# B&R Automation Studio project work
Automation Studio 4.5.2.102

## Configuration Config1

### Task classes (Cpu.sw)
```
Cyclic#1:
  Program <- Program.prg
Binaries: udbdef, TCData, iomap, ashwac, Role, sysconf, arconfig, asfw, User, ashwd
Libraries: Library1
```

## Logical view

Binary libraries used (declarations not repeated): operator, runtime, astime, AsIecCon

### Library Logical/Libraries/Library1 (ANSIC)

#### Library1.fun - Exported functions and function blocks
```iecst
{REDUND_ERROR} FUNCTION_BLOCK FB_Motor (*Функциональный блок для моделирования двигателя*) (*$GROUP=User,$CAT=User,$GROUPICON=User.png,$CATICON=User.png*)
	VAR_INPUT
		u : {REDUND_UNREPLICABLE} REAL;
	END_VAR
	VAR
		dt : REAL;
	END_VAR
	VAR_OUTPUT
		w : {REDUND_UNREPLICABLE} REAL;
		phi : {REDUND_UNREPLICABLE} REAL;
	END_VAR
	VAR
		integrator : {REDUND_UNREPLICABLE} FB_Integrator;
		Tm : {REDUND_UNREPLICABLE} REAL;
		ke : {REDUND_UNREPLICABLE} REAL;
	END_VAR
END_FUNCTION_BLOCK

{REDUND_ERROR} FUNCTION_BLOCK FB_Integrator (*Функциональный блок интегратора*) (*$GROUP=User,$CAT=User,$GROUPICON=User.png,$CATICON=User.png*)
	VAR_INPUT
		in : {REDUND_UNREPLICABLE} REAL;
	END_VAR
	VAR
		dt : REAL;
	END_VAR
	VAR_OUTPUT
		out : {REDUND_UNREPLICABLE} REAL;
	END_VAR
	VAR
		prev_value : REAL;
	END_VAR
END_FUNCTION_BLOCK

{REDUND_ERROR} FUNCTION_BLOCK FB_Controller (*TODO: Add your comment here*) (*$GROUP=User,$CAT=User,$GROUPICON=User.png,$CATICON=User.png*)
	VAR
		dt : REAL; (*шаг расчёта 0.01*)
	END_VAR
	VAR_INPUT
		e_in : {REDUND_UNREPLICABLE} REAL;
	END_VAR
	VAR_OUTPUT
		u_out : {REDUND_UNREPLICABLE} REAL;
	END_VAR
	VAR
		sum : REAL;
		a : REAL;
		k_p : REAL;
		k_i : REAL;
		max_abs_value : REAL;
		iyOld : REAL;
		integrator : FB_Integrator;
	END_VAR
END_FUNCTION_BLOCK
```

#### FB_Motor.c
```c
#include <bur/plctypes.h>
#ifdef __cplusplus
	extern "C"
	{
#endif
	#include "Library1.h"
#ifdef __cplusplus
	};
#endif
/* Функциональный блок для моделирования двигателя */
void FB_Motor(struct FB_Motor* inst)
{

	REAL a = inst->u/inst->ke - inst->w;
	REAL b = a / inst->Tm;

	inst->integrator.in = b;
	FB_Integrator(&inst->integrator);

	inst->w = inst->integrator.out;

}
```

#### FB_Integrator.c
```c
#include <bur/plctypes.h>
#ifdef __cplusplus
	extern "C"
	{
#endif
	#include "Library1.h"
#ifdef __cplusplus
	};
#endif
/* Функциональный блок интегратора */
void FB_Integrator(struct FB_Integrator* inst)
{
	inst->dt = d_t;
	inst->out = inst->dt * inst->in + inst->prev_value;
	inst->prev_value = inst->out;
}
```

#### FB_Controller.c
```c
#include <bur/plctypes.h>
#ifdef __cplusplus
	extern "C"
	{
#endif
	#include "Library1.h"
#ifdef __cplusplus
	};
#endif
/* TODO: Add your comment here */
void FB_Controller(struct FB_Controller* inst)
{
	REAL a = inst->e_in * inst->k_p;
	REAL b = inst->e_in * inst->k_i;

	a = a > inst->max_abs_value ? inst->max_abs_value : a;
	a = a < -inst->max_abs_value ? -inst->max_abs_value : a;

	inst->integrator.in = b + inst->iyOld;
	FB_Integrator(&inst->integrator);

	REAL sum = a + inst->integrator.out;

	inst->u_out = sum;
	inst->u_out = inst->u_out > inst->max_abs_value ? inst->max_abs_value : inst->u_out;
	inst->u_out = inst->u_out < -inst->max_abs_value ? -inst->max_abs_value : inst->u_out;
	inst->iyOld = inst->u_out - sum;

}
```

### Program Logical/Program

#### Variables.var
```iecst
VAR
	fb_motor1 : FB_Motor;
	fb_motor2 : FB_Motor;
	fb_controller : FB_Controller;
	enable : BOOL;
	counter : UINT;
	speed : REAL;
	fb_integrator1 : FB_Integrator;
END_VAR
```

#### Main.c
```c
#include <bur/plctypes.h>

#ifdef _DEFAULT_INCLUDES
	#include <AsDefault.h>
#endif

void _INIT ProgramInit(void)
{
	fb_motor1.ke = 0.24;
	fb_motor1.Tm = 0.1;
	fb_motor1.u = 0;

	fb_motor2.ke = 0.24;
	fb_motor2.Tm = 0.1;
	fb_motor2.u = 0;

	fb_controller.k_p = 0.24*3;
	fb_controller.k_i = 7.2;
	fb_controller.max_abs_value = 24.0;
	fb_controller.dt = 0.01;
	fb_controller.integrator.dt=0.001;

	speed = 0;
	counter = 0;
	enable = 1;

}

void _CYCLIC ProgramCyclic(void)
{
	if(enable)
	{

		if(counter == 200)
		{
			speed = 50;
		}
		else if (counter == 400)
		{
			speed = 0;
			counter= 0;
		}

		counter++;

		fb_controller.e_in = speed - fb_motor1.w;
		FB_Controller(&fb_controller);

		fb_motor1.u = fb_controller.u_out;

		fb_motor2.u = speed * fb_motor2.ke;

		FB_Motor(&fb_motor1);
		FB_Motor(&fb_motor2);

		fb_integrator1.in = fb_motor1.w;
		FB_Integrator (&fb_integrator1);
	}
}

void _EXIT ProgramExit(void)
{

}
```

Listed in the project but not available here: Logical/Libraries/Library1/Types.typ, Logical/Libraries/Library1/Constants.var
